PROGRAM BroadcastExample
VAR
END_VAR

SafetyExample();

END_PROGRAM

(* stored: Version 1.1.0.1
   POU BroadcastExample: Id {eeeb7f20-33e5-4527-bff4-eb13d57b2084}, SpecialFunc None *)
